(* Logix 5000 project; controller Ex_2_11 Emulate 5570 rev 33.11; software revision 33.00 *)
// Pacakge on conveyor belt

TASK MainTask (continuous, watchdog 500 ms) : MainProgram

MODULES
   Local : Emulate 5570 (ICP 4, rev 33.11)
END_MODULES

PROGRAM MainProgram   (* main routine MainRoutine *)

ROUTINE MainRoutine   (* ladder *)
END_ROUTINE
END_PROGRAM
